FUNCTION_BLOCK ConvCtrl
  (* Standard: 61499-2 *)
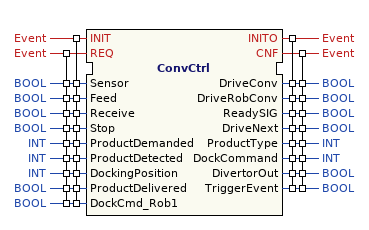
  EVENT_INPUT
    INIT WITH Sensor, Feed, Receive, Stop, ProductDemanded, ProductDetected, DockingPosition, ProductDelivered, DockCmd_Rob1;
    REQ WITH Sensor, Feed, Receive, Stop, ProductDemanded, ProductDetected, DockingPosition, ProductDelivered, DockCmd_Rob1;
  END_EVENT
  EVENT_OUTPUT
    INITO WITH DriveConv, DriveRobConv, ReadySIG, DriveNext, ProductType, DockCommand, DivertorOut, TriggerEvent;
    CNF WITH DriveConv, DriveRobConv, ReadySIG, DriveNext, ProductType, DockCommand, DivertorOut, TriggerEvent;
  END_EVENT
  VAR_INPUT
    Sensor : BOOL;
    Feed : BOOL;
    Receive : BOOL;
    Stop : BOOL;
    ProductDemanded : INT;
    ProductDetected : INT;
    DockingPosition : INT;
    ProductDelivered : BOOL;
    DockCmd_Rob1 : BOOL;
  END_VAR
  VAR_OUTPUT
    DriveConv : BOOL;
    DriveRobConv : BOOL;
    ReadySIG : BOOL;
    DriveNext : BOOL;
    ProductType : INT;
    DockCommand : INT;
    DivertorOut : BOOL;
    TriggerEvent : BOOL;
  END_VAR
  VAR
    TimeStamp : DATE_AND_TIME;
  END_VAR
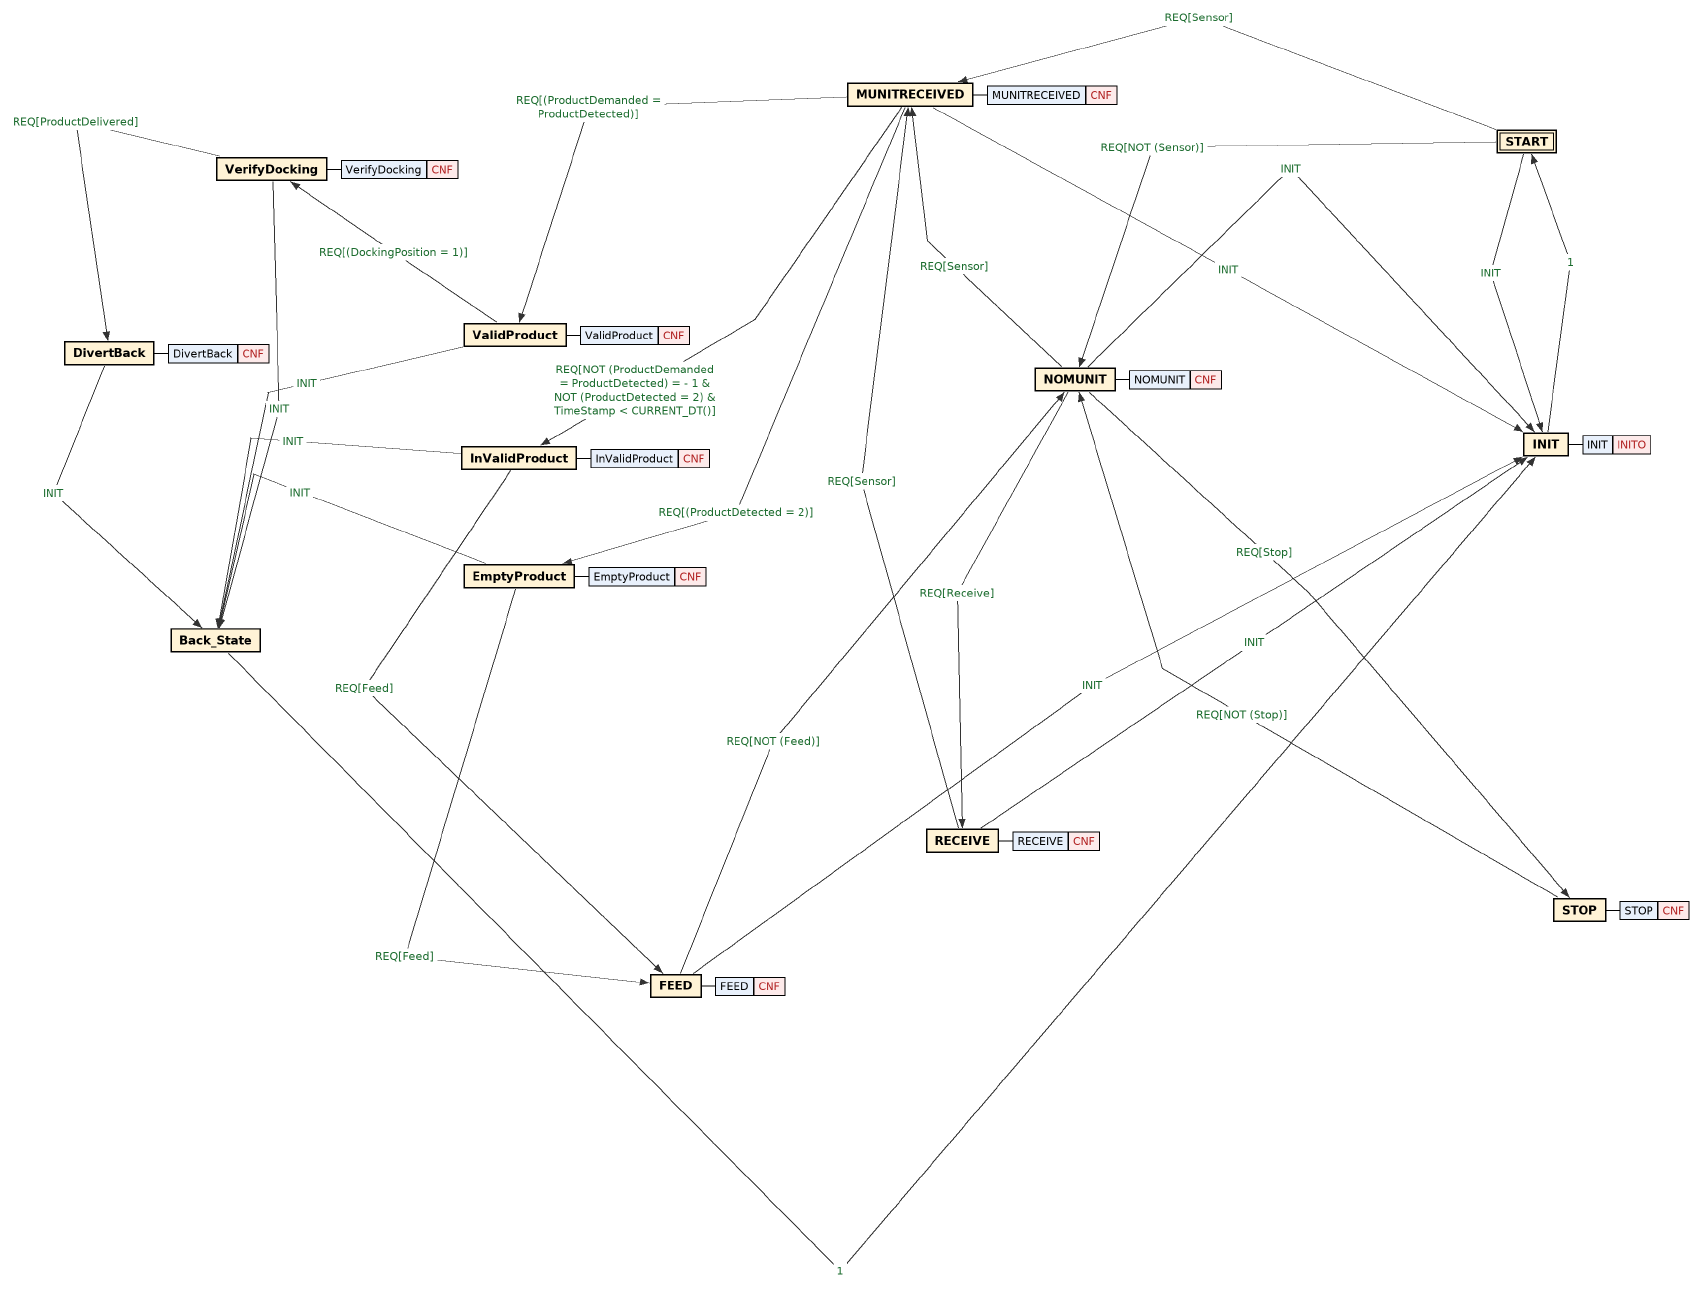
  EC_STATES
    START;
    INIT : INIT -> INITO;
    FEED : FEED -> CNF;
    MUNITRECEIVED : MUNITRECEIVED -> CNF;
    NOMUNIT : NOMUNIT -> CNF;
    RECEIVE : RECEIVE -> CNF;
    STOP : STOP -> CNF;
    ValidProduct : ValidProduct -> CNF;
    InValidProduct : InValidProduct -> CNF;
    EmptyProduct : EmptyProduct -> CNF;
    Back_State;
    VerifyDocking : VerifyDocking -> CNF;
    DivertBack : DivertBack -> CNF;
  END_STATES
  EC_TRANSITIONS
    START TO INIT := INIT;
    INIT TO START := 1;
    NOMUNIT TO MUNITRECEIVED := REQ[Sensor];
    FEED TO NOMUNIT := REQ[NOT (Feed)];
    RECEIVE TO MUNITRECEIVED := REQ[Sensor];
    START TO MUNITRECEIVED := REQ[Sensor];
    NOMUNIT TO RECEIVE := REQ[Receive];
    START TO NOMUNIT := REQ[NOT (Sensor)];
    RECEIVE TO INIT := INIT;
    NOMUNIT TO INIT := INIT;
    FEED TO INIT := INIT;
    MUNITRECEIVED TO INIT := INIT;
    NOMUNIT TO STOP := REQ[Stop];
    STOP TO NOMUNIT := REQ[NOT (Stop)];
    MUNITRECEIVED TO ValidProduct := REQ[(ProductDemanded = ProductDetected)];
    MUNITRECEIVED TO InValidProduct := REQ[NOT (ProductDemanded = ProductDetected) = - 1 & NOT (ProductDetected = 2) & TimeStamp < CURRENT_DT()];
    MUNITRECEIVED TO EmptyProduct := REQ[(ProductDetected = 2)];
    InValidProduct TO Back_State := INIT;
    EmptyProduct TO Back_State := INIT;
    InValidProduct TO FEED := REQ[Feed];
    EmptyProduct TO FEED := REQ[Feed];
    Back_State TO INIT := 1;
    ValidProduct TO VerifyDocking := REQ[(DockingPosition = 1)];
    VerifyDocking TO Back_State := INIT;
    ValidProduct TO Back_State := INIT;
    VerifyDocking TO DivertBack := REQ[ProductDelivered];
    DivertBack TO Back_State := INIT;
  END_TRANSITIONS
  ALGORITHM INIT IN ST:
DriveConv := 0;&#10;ReadySIG := 1;&#10;DriveNext := 0;&#10;ProductDetected := - 1;&#10;ProductType := - 1;&#10;
  END_ALGORITHM
  ALGORITHM FEED IN ST:
DriveConv := 1;&#10;ReadySIG := 0;&#10;DriveNext := 1;&#10;DivertorOut := 0;&#10;DriveRobConv := FALSE;&#10;TriggerEvent := FALSE;&#10;
  END_ALGORITHM
  ALGORITHM MUNITRECEIVED IN ST:

  END_ALGORITHM
  ALGORITHM NOMUNIT IN ST:

  END_ALGORITHM
  ALGORITHM RECEIVE IN ST:
DriveConv := 1;&#10;ReadySIG := 1;&#10;DriveNext := 0;&#10;DivertorOut := 0;&#10;DriveRobConv := FALSE;&#10;TriggerEvent := FALSE;&#10;
  END_ALGORITHM
  ALGORITHM STOP IN ST:
DriveConv := 0;&#10;ReadySIG := 0;&#10;DriveNext := 0;&#10;DivertorOut := 0;&#10;DriveRobConv := FALSE;&#10;TriggerEvent := FALSE;&#10;
  END_ALGORITHM
  ALGORITHM ValidProduct IN ST:

  END_ALGORITHM
  ALGORITHM InValidProduct IN ST:

  END_ALGORITHM
  ALGORITHM EmptyProduct IN ST:

  END_ALGORITHM
  ALGORITHM VerifyDocking IN ST:

  END_ALGORITHM
  ALGORITHM DivertBack IN ST:

  END_ALGORITHM
END_FUNCTION_BLOCK
